INTERFACE I_Module

{attribute 'monitoring' := 'call'}
PROPERTY bEstop : BOOL
GET
END_GET
SET
END_SET
END_PROPERTY

{attribute 'monitoring' := 'call'}
PROPERTY bSleep : BOOL
GET
END_GET
SET
END_SET
END_PROPERTY

(*
  Register to get Emergency state updates.
*)
METHOD registerForEmergencyUpdate : BOOL
VAR_INPUT
	iObserver	: I_EmergencyObserver;
END_VAR
END_METHOD

(*
  Register to get sleep state updates.
*)
METHOD registerForSleepUpdate : BOOL
VAR_INPUT
	iObserver	: I_SleepObserver;
END_VAR
END_METHOD

END_INTERFACE

(* stored: Version 1.1.0.1, ProductVersion 3.1.4024.11
   Itf I_Module: Id {1dfd1863-e2a6-441a-9d89-aba8aeeb8a6a}
   Property bEstop: Id {4b1b4922-80a7-423d-9cfc-b78fbc2175c5}
   Get Get: Id {0c7d3028-0d52-4087-a8eb-f2b7d6c2ba3e}
   Set Set: Id {e277afc3-0577-4eb6-abeb-41eed3168691}
   Property bSleep: Id {47e04413-cad2-427c-b47f-a7499a7b8296}
   Get Get: Id {39547459-ada4-423c-9e42-25550573bb7e}
   Set Set: Id {922ce03d-1716-4fec-831d-71336752c26f}
   Method registerForEmergencyUpdate: Id {5e2c4080-670f-4c98-96bf-407b75d7c2b3}
   Method registerForSleepUpdate: Id {1f9b7c9c-a46b-4be8-9d82-e785f6af3470} *)
